FUNCTION AVG (* Array Average *)
  (* Standard: 61499-1 *)
  (* Version 1.0, 2026-01-23, Franz Höpfinger, Andreas Demmler Fahrzeugbau, inspired by AVG in IEC 61131 Paper *)
  PACKAGE logiBUS::utils::dyn_arr;
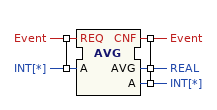
  EVENT_INPUT
    REQ WITH A;
  END_EVENT
  EVENT_OUTPUT
    CNF WITH AVG, A;
  END_EVENT
  VAR_OUTPUT
    AVG : REAL;
  END_VAR
  VAR_IN_OUT
    A : ARRAY [*] OF INT; (* Input *)
  END_VAR
  BODY IN ST:
PACKAGE logiBUS::utils::dyn_arr;

(* Array Average *)
FUNCTION AVG : REAL

VAR_IN_OUT
	A : ARRAY[*] OF INT; // Input
END_VAR

VAR_TEMP
	i : INT;
	sum : DINT;
	count : INT;
END_VAR

sum := 0;

FOR i := LOWER_BOUND(A,1) TO UPPER_BOUND(A,1) DO
	sum := sum + A[i];
END_FOR;
count := UPPER_BOUND(A, 1) - LOWER_BOUND(A, 1) + 1;
AVG := DINT_TO_REAL(sum) / INT_TO_REAL(count);

END_FUNCTION
  END_BODY
END_FUNCTION
